PROGRAM Ladder
VAR

END_VAR
VAR // added by the converter: edge detectors and wires of the graphical bodies
    _rt1 : R_TRIG;
END_VAR

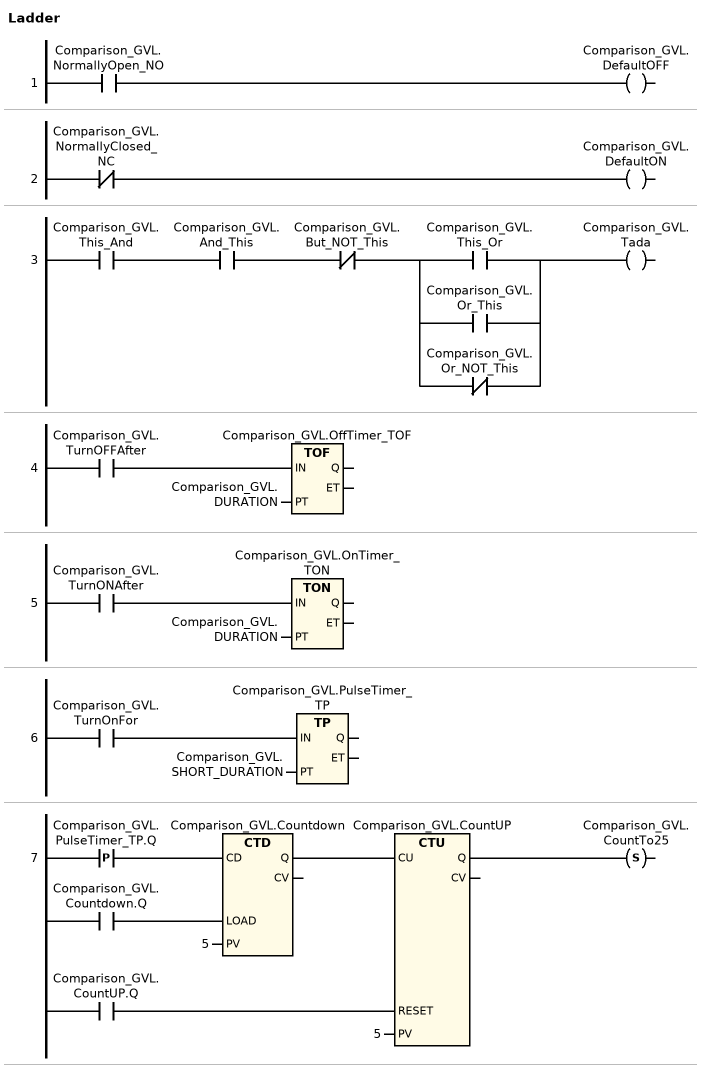
// NETWORK 1
Comparison_GVL.DefaultOFF := Comparison_GVL.NormallyOpen_NO;

// NETWORK 2
Comparison_GVL.DefaultON := NOT Comparison_GVL.NormallyClosed_NC;

// NETWORK 3
Comparison_GVL.Tada := Comparison_GVL.This_And AND Comparison_GVL.And_This AND NOT Comparison_GVL.But_NOT_This AND (Comparison_GVL.This_Or OR Comparison_GVL.Or_This OR NOT Comparison_GVL.Or_NOT_This);

// NETWORK 4
Comparison_GVL.OffTimer_TOF(IN := Comparison_GVL.TurnOFFAfter, PT := Comparison_GVL.DURATION); // TOF

// NETWORK 5
Comparison_GVL.OnTimer_TON(IN := Comparison_GVL.TurnONAfter, PT := Comparison_GVL.DURATION); // TON

// NETWORK 6
Comparison_GVL.PulseTimer_TP(IN := Comparison_GVL.TurnOnFor, PT := Comparison_GVL.SHORT_DURATION); // TP

// NETWORK 7
_rt1(CLK := Comparison_GVL.PulseTimer_TP.Q);
Comparison_GVL.Countdown(CD := _rt1.Q, LOAD := Comparison_GVL.Countdown.Q, PV := 5); // CTD
Comparison_GVL.CountUP(CU := Comparison_GVL.Countdown.Q, RESET := Comparison_GVL.CountUP.Q, PV := 5); // CTU
Comparison_GVL.CountTo25 S= Comparison_GVL.CountUP.Q;

END_PROGRAM

(* stored: Version 1.1.0.1, ProductVersion 3.1.4024.11
   POU Ladder: Id {dfbb198f-7d9c-4f2c-9ba5-fdf48be9a7a9}, SpecialFunc None *)
